// TIA Portal V17 export
// export: Created 2025-03-05T08:01:13.346927Z, ExportSetting WithDefaults, DisplayName Totally Integrated Automation Portal, DisplayVersion V17 Update 8, DisplayName TIA Portal Openness, DisplayVersion V17 Update 8, DisplayName TIA Portal Version Control Interface, DisplayVersion V17, DisplayName SINAMICS Startdrive Advanced, DisplayVersion V17 SP2, DisplayName SINAMICS Startdrive G110M, G120, G120C, G120D, G120P, G115D, DisplayVersion V17 SP2, DisplayName SINAMICS Startdrive G130, G150, S120, S150, SINAMICS MV, S210, DisplayVersion V17 SP2, DisplayName STEP 7 Professional, DisplayVersion V17 Update 8, DisplayName SINUMERIK ONE STEP 7 Toolbox, DisplayVersion V17 Update 12, DisplayName SINUMERIK 840D sl STEP 7 Toolbox, DisplayVersion V17 Update 12, DisplayName STEP 7 Safety, DisplayVersion V17 Update 6, DisplayName WinCC Advanced, DisplayVersion V17 Update 8
DATA_BLOCK "DB2203_PROFINET_INSPEKTOR"   // DB2203
{ S7_Optimized_Access := 'FALSE'; DB_Accessible_From_OPC_UA := 'FALSE' }
VERSION : 0.1
// stored: AutoNumber false, DBAccessibleFromOPCUA false, DBAccessibleFromWebserver true, IsOnlyStoredInLoadMemory false, IsWriteProtectedInAS false
   VAR
      PROFINET_FAULT_I : Bool;   // PROFINET INSPEKTOR PROFINET FAULT INPUT
      SPARE_01 : Bool;   // SPARE 01
      SPARE_02 : Bool;   // SPARE 02
      SPARE_03 : Bool;   // SPARE 03
      PROFINET_FAULT_PRESENT : Bool;   // PROFINET INSPEKTOR PROFINET FAULT PRESENT
      SPARE_05 : Bool;   // SPARE 05
      SPARE_06 : Bool;   // SPARE 06
      SPARE_07 : Bool;   // SPARE 07
      PFI_ACKNOW_FAULTS_IMPULS : Bool;   // PROFINET INSPEKTOR ACKOWLEDGE FAULTS IMPULSE
      SPARE_11 : Bool;   // SPARE 11
      SPARE_12 : Bool;   // SPARE 12
      SPARE_13 : Bool;   // SPARE 13
      SPARE_14 : Bool;   // SPARE 14
      SPARE_15 : Bool;   // SPARE 15
      SPARE_16 : Bool;   // SPARE 16
      PFI_FAULTS_GONE : Bool;   // PROFINET INSPEKTOR FAULTS GONE
      PFI_START_Q : Bool;   // PROFINET INSPEKTOR START OUTPUT
      PFI_ACKNOWLEDGE_FAULTS_Q : Bool;   // PROFINET INSPEKTOR ACKOWLEDGE FAULTS OUTPUT
      PFI_DELETE_LOGGED_DATA_Q : Bool;   // PROFINET INSPEKTOR LOGGED DATA OUTPUT
      TIMER_ON_PFI_ACK_FAULTS_IMPULSE : TON_TIME;
      TIMER_OFF_PFI_ACK_FAULTS_IMPULSE : TOF_TIME;
      TIMER_ON_PFI_PROFINET_FAULT_PRESENT : TON_TIME;
   END_VAR
BEGIN
   TIMER_ON_PFI_ACK_FAULTS_IMPULSE.PT := T#5s;
   TIMER_OFF_PFI_ACK_FAULTS_IMPULSE.PT := T#2s;
   TIMER_ON_PFI_PROFINET_FAULT_PRESENT.PT := T#5s;
END_DATA_BLOCK
